Universal Robots PolyScope program: motor_plate_positioning_a_bot.urp

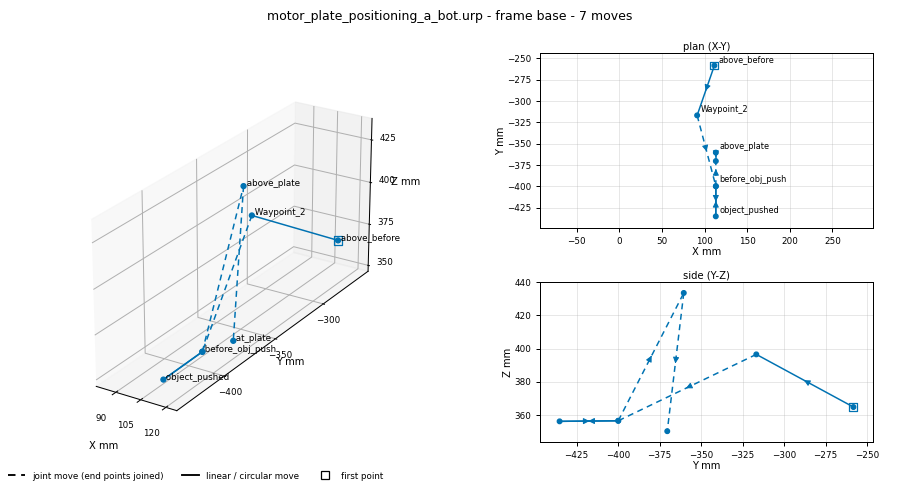
[picture p0: tool path of motor_plate_positioning_a_bot.urp in frame base, 7 of 8 moves have a stored position in this frame; points joined in program order, loops and branches not executed]
Program motor_plate_positioning_a_bot (installation=default directory=/programs createdIn=5.6.0.90886 lastSavedIn=5.6.0.90886 robotSerialNumber=20205500180)
Calibrated DH parameters: a=[0.000135, -0.030981, -0.334292, 0.000083, 0.000088, 0]; d=[0.162656, 258.79096, -331.603246, 72.945842, 0.099724, 0.099562]; alpha=[1.569535, 0.001639, 0.002824, 1.569633, -1.569323, 0]; deltaTheta=[0, 1.497881, -2.049261, 0.551379, 0, 0]
Robot Program (runOnlyOnce=true)
  MoveL speed 250 mm/s, acceleration 1200 mm/s^2 (useActiveTCP=true) feature=Base
    Waypoint Waypoint_1 (Relative): relativeFromPosition TCP in base x=111.497 y=-274.795 z=272.984 mm, rx=0 ry=-2.7207 rz=1.5708 rad; joints [83.27, -108.613, 132.077, 6.618, 84.039, 176.688] deg; TCP in base x=111.507 y=-258.31 z=272.993 mm, rx=0 ry=2.7207 rz=-1.5708 rad; joints [82.569, -111.657, 133.893, 7.884, 83.423, 176.326] deg
  URCap Gripper (Robotiq_Grippers, Robotiq Inc.) dataModel(position=72.54901960784314, force=0.0, speed=0.0, positionInDouble=72.54901960784314, forceInDouble=0.0, speedInDouble=0.0, slaveIds=[9], blocking=true)
  MoveL speed 250 mm/s, acceleration 1200 mm/s^2 (useActiveTCP=true) feature=Base
    Waypoint above_before: TCP in base x=111.502 y=-258.323 z=364.836 mm, rx=0 ry=-2.7207 rz=1.5708 rad; joints [82.551, -115.589, 122.176, 23.536, 83.376, 176.279] deg
    Waypoint Waypoint_2: TCP in base x=91.263 y=-316.792 z=396.54 mm, rx=1.7852 ry=-1.046 rz=2.1789 rad; joints [61.544, -119.489, 127.001, -32.837, 7.938, 140.093] deg
    MoveJ speed 60 deg/s, acceleration 80 deg/s^2 (useActiveTCP=true) feature=Base
      Waypoint before_obj_push: TCP in base x=113.226 y=-399.906 z=356.565 mm, rx=0.004 ry=3.141 rz=0.0154 rad; joints [87.172, -100.511, 118.783, -107.626, -89.818, -2.678] deg
  URCap Gripper (Robotiq_Grippers, Robotiq Inc.) dataModel(position=100.0, force=0.0, speed=0.0, positionInDouble=100.0, forceInDouble=0.0, speedInDouble=0.0, slaveIds=[9], blocking=true)
  MoveL speed 250 mm/s, acceleration 1200 mm/s^2 (useActiveTCP=true) feature=Base
    Waypoint object_pushed: motionParameters(jointSpeed=1.047198 jointAcceleration=1.396263 cartesianSpeed=0.008 cartesianAcceleration=1.2); TCP in base x=113.139 y=-435.23 z=356.222 mm, rx=0.004 ry=3.141 rz=0.0154 rad; joints [87.384, -95.381, 114.516, -108.489, -89.814, -2.455] deg
    Waypoint before_obj_push: TCP in base x=113.226 y=-399.906 z=356.565 mm, rx=0.004 ry=3.141 rz=0.0154 rad; joints [87.172, -100.511, 118.783, -107.626, -89.818, -2.678] deg
  URCap Gripper (Robotiq_Grippers, Robotiq Inc.) dataModel(position=72.54901960784314, force=0.0, speed=0.0, positionInDouble=72.54901960784314, forceInDouble=0.0, speedInDouble=0.0, slaveIds=[9], blocking=true)
  MoveJ speed 60 deg/s, acceleration 80 deg/s^2 (useActiveTCP=true) feature=Base
    Waypoint above_plate: TCP in base x=113.193 y=-360.458 z=433.533 mm, rx=0.0037 ry=3.0617 rz=-0.699 rad; joints [86.404, -112.982, 123.786, -126.397, -88.216, -3.05] deg
    Waypoint at_plate: TCP in base x=113.193 y=-370.401 z=350.29 mm, rx=0.0037 ry=3.0617 rz=-0.699 rad; joints [86.494, -106.791, 132.85, -141.656, -88.265, -2.917] deg
  URCap Gripper (Robotiq_Grippers, Robotiq Inc.) dataModel(position=100.0, force=0.0, speed=0.0, positionInDouble=100.0, forceInDouble=0.0, speedInDouble=0.0, slaveIds=[9], blocking=true)
